// TIA Portal V17 export
// export: Created 2025-06-26T06:33:55.7435126Z, ExportSetting WithDefaults, DisplayName Totally Integrated Automation Portal, DisplayVersion V17 Update 8, DisplayName TIA Portal Openness, DisplayVersion V17 Update 8, DisplayName TIA Portal Version Control Interface, DisplayVersion V17, DisplayName STEP 7 Professional, DisplayVersion V17 Update 8, DisplayName STEP 7 Safety, DisplayVersion V17 Update 6, DisplayName WinCC Advanced, DisplayVersion V17 Update 8
DATA_BLOCK "Customer_DB"   // DB11
AUTHOR : Heaten
VERSION : 0.1
// stored: AutoNumber true, DBAccessibleFromOPCUA true, InstanceOfName Customer, InstanceOfType FB
"Customer"
   // VAR
   //    Watchdog { S7_SetPoint := 'True'} : "fbHeartbeatCount2";
   //    epStartRequest { S7_SetPoint := 'True'} : Bool;
   //    enStartRequest : Bool;
   //    epStopRequest : Bool;
   //    enStopRequest : Bool;
   //    epAlarmAcknowledge : Bool;
   //    enAlarmAcknowledge : Bool;
   //    epResetEmergencyStop : Bool;
   //    enResetEmergencyStop : Bool;
   //    SetpointPrev : Real;
   //    RegulationTargetPrev : Int;
   //    HCV812Cmd : Real;
   //    HCV815Cmd : Real;
   //    HCV818Cmd : Real;
   //    HCV821Cmd : Real;
   // END_VAR
BEGIN
END_DATA_BLOCK
